// TwinCAT 3 PLC project ThermalControl_PLC
// ProgramVersion: 3.1.4023.0
// libraries:
//   Tc2_ControllerToolbox, * (Beckhoff Automation GmbH)
//   Tc2_Standard, * (Beckhoff Automation GmbH)
//   Tc2_System, * (Beckhoff Automation GmbH)
//   Tc2_TempController, * (Beckhoff Automation GmbH)
//   Tc3_Module, * (Beckhoff Automation GmbH)
// project tree:
//   / Cyclic100ms.TcTTO (not stored), PlcTask.TcTTO
//   DUTs/ E_State.TcDUT (not stored), ST_ThermalCouple.TcDUT (not stored)
//   GVLs/ GVL.TcGVL, HMI_DB.TcGVL (not stored), Input.TcGVL, MCP_IO.TcGVL (not stored), Output.TcGVL
//   POUs/ ADC_10V.TcPOU (not stored), ADC_5V.TcPOU (not stored), Alias.TcPOU, AnalogConversion.TcPOU (not stored), AQ.TcPOU (not stored), AQ_5V.TcPOU, FB_Process.TcPOU, Heartbeat.TcPOU (not stored), MAIN.TcPOU (not stored), Norm_x.TcPOU (not stored), Sequence.TcPOU
//   POUs/Controller/ Controller_v1.TcPOU, Controller_v2.TcPOU (not stored)
//   POUs/PID/ PRG_FB_CTRL_PID.TcPOU

CONFIGURATION ThermalControl_PLC
    RESOURCE PLC ON TwinCAT3
        TASK PlcTask(INTERVAL := T#10ms, PRIORITY := 20);
        PROGRAM MAIN WITH PlcTask : MAIN;
    END_RESOURCE
END_CONFIGURATION

// ---- GVLs/GVL.TcGVL
{attribute 'qualified_only'}
VAR_GLOBAL
	SetpointValueToScope			: LREAL;
	ActualValueToScope				: LREAL;
	OutToScope						: LREAL;
END_VAR

// ---- GVLs/Input.TcGVL
{attribute 'qualified_only'}
VAR_GLOBAL
//***MCP************************************************************************
	//EL3314 - AI1
	R1_01_00 AT	%I*: INT; //Master stop PB not pressed - black pb on mcp
	R1_01_01 AT	%I*: INT; //case Estop circuit okay (Rly1 (120vac)
	R1_01_02 AT %I*: INT; //Remote Mode Selected (NO)
	R1_01_03 AT %I*: INT; //MCP PSU1 DC OK
	
	//EL3314 - AI2
	R1_02_00 AT	%I*: INT; //
	R1_02_01 AT	%I*: INT;
	R1_02_02 AT %I*: INT; 
	R1_02_03 AT %I*: INT; 
	
	//EL3314 - AI3
	R1_03_00 AT	%I*: INT; //
	R1_03_01 AT	%I*: INT;
	R1_03_02 AT %I*: INT; 
	R1_03_03 AT %I*: INT; 

END_VAR

// ---- GVLs/Output.TcGVL
{attribute 'qualified_only'}
VAR_GLOBAL
	//***MCP 
	//EL2008
	R1_13_00 AT %Q*: BOOL;
	
	//EL4008 - AQ1
	R1_18_00 AT %Q*: INT;
	R1_18_01 AT %Q*: INT;
	R1_18_02 AT %Q*: INT;
	R1_18_03 AT %Q*: INT;
	R1_18_04 AT %Q*: INT;
	R1_18_05 AT %Q*: INT;
	R1_18_06 AT %Q*: INT;
	R1_18_07 AT %Q*: INT;

	
END_VAR

// ---- POUs/Alias.TcPOU
PROGRAM Alias
VAR
	i : INT := 0;
END_VAR

 //R1 : MCP**  
	
//INPUT
	//AI	
	MCP_IO.ThermalCouple[1].Temperature_raw					:= Input.R1_01_00;  //NC -
	MCP_IO.ThermalCouple[2].Temperature_raw					:= Input.R1_01_01;  
	MCP_IO.ThermalCouple[3].Temperature_raw					:= Input.R1_01_02; 
	MCP_IO.ThermalCouple[4].Temperature_raw					:= Input.R1_01_03; 

	MCP_IO.ThermalCouple[5].Temperature_raw					:= Input.R1_02_00;  //NC -
	MCP_IO.ThermalCouple[6].Temperature_raw					:= Input.R1_02_01;  
	MCP_IO.ThermalCouple[7].Temperature_raw					:= Input.R1_02_02; 
	MCP_IO.ThermalCouple[8].Temperature_raw					:= Input.R1_02_03; 
	
	MCP_IO.ThermalCouple[9].Temperature_raw					:= Input.R1_03_00;  //NC -
	MCP_IO.ThermalCouple[10].Temperature_raw				:= Input.R1_03_01;  
	MCP_IO.ThermalCouple[11].Temperature_raw				:= Input.R1_03_02; 
	MCP_IO.ThermalCouple[12].Temperature_raw				:= Input.R1_03_03; 
	
	//OUTPUT
	//AQ
	Output.R1_18_00	:= MCP_IO.ChargerSP_raw;
					
	

	
//*************************************************************************************************************

END_PROGRAM

// ---- POUs/AQ_5V.TcPOU
FUNCTION AQ_5V : INT
VAR_INPUT
	Norm_input : REAL;
	x_max : REAL := 10;
	x_min : REAL := 0;
END_VAR
VAR
	voltage_reading : REAL;
END_VAR

voltage_reading := 5 * Norm_input;
AQ_5V := REAL_TO_INT (32767 * (voltage_reading - x_min) / (x_max - x_min));

END_FUNCTION

// ---- POUs/Controller/Controller_v1.TcPOU
PROGRAM Controller_v1

VAR
	
	bOn						: BOOL	:= TRUE;
	bSelSetpoint 			: BOOL	:= FALSE;
	bInit					: BOOL 	:= TRUE;
	bTune					: BOOL 	:= TRUE;
	bManual					: BOOL;

	bNoise 					: BOOL;
	bError 					: BOOL;
	iErrorId 				: E_ErrorCodes;

	fW						: LREAL;						(* setpoint *)
	fW1						: LREAL := 	70;					(* first setpoint *)
	fW2						: LREAL :=	35.0;				(* second setpoint - standby setpoint*)
	fY						: LREAL;						(* control value *)
	fX						: LREAL;						(* actual value from simulated process *)
	bYPWM					: BOOL;

	bSelParameterSet		: BOOL := FALSE;
	bEnableSoftStart 		: BOOL := TRUE;
	bEnableRamping 			: BOOL := FALSE;

	(* parameters *)
	sControllerParameter	:	ST_ControllerParameter := ( 	
	
	iMode 					:= CTRLMODE_HEATING, 							(* 1=heating, 2=cooling, 3=heating&cooling *)
	iReactionOnFailure 		:= TC_OnFailureStopController,					(* 0=controller off, 1=manual op, 2=yMin, 3=yMax *)
	
	dwAlarmSupp 			:= 16#FF_FF_FF_FF, 								(* alarm suppression *)
	tCtrlCycleTime 			:= T#500MS, 									(* controller cycle time *)
	tTaskCycleTime 			:= T#10MS,										(* plc task cycle time *)
	fYTune 					:= 100.0,										(* switch to closed loop control when X > 0.8*W *)
	
	tPWMCycleTime 			:= T#40MS,										(* PWM: period *)
	
	(* setpoint parameters 													 *)	
	fWMin 					:= 0, 											(* lower limit *)
	fWMax 					:= 300,  										(* upper limit *)
	
	(* start up 															*)
	fWStartUp 				:= 0.0, //40.0,									(* soft start plateau setpoint *)
	tStartUp 				:= T#0MS,// T#20S,								(* soft start waiting time*)
 	bStartUpRamping 		:= FALSE,//TRUE, 								(* enable ramping while start up phase *)
	fWStartUpVeloPos 		:= 1.0, 										(* max gradient for increasing setpoint in start up phase*)
	fWStartUpVeloNeg 		:= 1.0,											(* max gradient for decreasing setpoint in start up phase*)
	
	fWVeloPos 				:= 1.0,											(* max gradient for increasing setpoint *) 
	fWVeloNeg 				:= 1.0,											(* max gradient for decreasing setpoint *)	
	
	(* actual value parameters     											 *)	
	bFilter 				:= FALSE, 	
	tFilter 				:= T#0S,
	
	(* control value parameters     										 *)
	fYMin 					:= 0.0, 										(* lower limit *)
	fYMax 					:= 100.0, 										(* upper limit *)
	fYManual 				:= 0.0,											(* manual operation*)
	
	(* controller settings			     									 *)
	bEnablePreController 	:= FALSE,										(* enable precontroller *)		
	bEnableZones 			:= FALSE, 										(* enable zone around setpoint with open loop control *)	
	bEnableCVFilter 		:= FALSE,	 									(* enable filter for CV (type see iFilterType) *)
	iFilterType 			:= E_FilterType_FIRSTORDER,						(* filtertype of CV filter *)
	iControllerType 		:= E_ControllerType_PID,						(* used controller normally PID *)
	
	(* min max temperatures	     											 *)
	TempLow 				:= -5.0, 
	TempLowLow 				:= -10.0,  
	TempHigh			 	:= 5.0, 
	TempHighHigh 			:= 10.0, 
	TempAbsoluteHigh 		:= 300.0, 
	TempAbsoluteLow 		:= 0.0
	
	);
								
	sParaControlExternal	: st_ParaController;
	
	fbTempController		: FB_TempController;
	fbProcess				: FB_Process;
	fbCtrlParameter			: FB_CtrlParameter;	
	
	(* Debug *)
	fMaxOvershoot			: LREAL;
	tStartUpTime			: TIME;
	eCtrlState				: E_CTRL_STATE;	
	
END_VAR

(* Select setpoint *)
IF bSelSetpoint THEN
	fW := fW2;
ELSE
	fW := fW1;
END_IF

(* Simulate process *)
fbProcess(	fY := fbTempController.fYAnalog, 
			bNoise := bNoise, 
			tTa := sControllerParameter.tTaskCycleTime);
			
(* Actual temperature *)				
fX := fbProcess.fX;  // Add measured temperature here

(* Start controller *)
fbTempController(
					bOn						:= bOn,
					bInit					:= bInit,
					bTune					:= bTune,
					bManual					:= bManual,
					bSelSetpoint			:= bSelSetpoint,
					bSelCtrlParameterSet 	:= bSelParameterSet,
					bEnableSoftStart 		:= bEnableSoftStart,
					bEnableRamping 			:= bEnableRamping,
					fW1						:= fW1,
					fW2						:= fW2,
					fX						:= fX,
					bOpenThermocouple		:= FALSE,
					bReverseThermocouple	:= FALSE,
					bBackVoltage			:= FALSE,
					bLeakage				:= FALSE,
					bShortCircuit			:= FALSE,
					bOpenCircuit			:= FALSE,
					sControllerParameter	:= sControllerParameter,
					sParaControllerExternal	:= fbCtrlParameter.sParaController
					);
					
(* Analog output *)			
fY := fbTempController.fYAnalog;
(* Digital (PWM) output *)
bYPWM := fbTempController.bYPWM;

bError := fbTempController.bError;
iErrorId := fbTempController.iErrorId;
bInit := FALSE;	

(* Debug *)
fMaxOvershoot := fbTempController.fMaxOverShoot;
tStartUpTime := fbTempController.tStartUpTime;

(* Scope *)
fW_Scope := fW;
fX_Scope := fX;
fY_Scope := fY;

END_PROGRAM

// ---- POUs/FB_Process.TcPOU
FUNCTION_BLOCK FB_Process

VAR_INPUT
	fY		:	LREAL;
	tTa		:	TIME;
	bNoise	:	BOOL;
END_VAR

VAR_OUTPUT
	fX		:	LREAL;
END_VAR

VAR
	(* Processparameters *)
	tT11		:	TIME	:= t#5s;
	tT12		:	TIME	:= t#25s;

	(* process *)
	fbProcessPart1	:	FB_CTRL_PT1;
	fbProcessPart2	:	FB_CTRL_PT1;
	fbNoise			:	FB_CTRL_NOISE_GENERATOR;

	stProcessPart1	:	ST_CTRL_PT1_PARAMS;
	stProcessPart2	:	ST_CTRL_PT1_PARAMS;
	stNoise			:	ST_CTRL_NOISE_GENERATOR_PARAMS;
	
END_VAR

(* init structures *)
stProcessPart1.fKp := 1.0;
stProcessPart1.tCtrlCycleTime := tTa;
stProcessPart1.tT1 := tT11;
stProcessPart1.tTaskCycleTime := tTa;

stProcessPart2.fKp := 1.0;
stProcessPart2.tCtrlCycleTime := tTa;
stProcessPart2.tT1 := tT12;
stProcessPart2.tTaskCycleTime := tTa;

stNoise.fAmplitude := 1.0;
stNoise.tCtrlCycleTime := tTa;
stNoise.tTaskCycleTime := tTa;

(* calculate and simulate process *)
fbProcessPart1(
				fIn:= fY,
				fManSyncValue:= 0.0,
				bSync:= FALSE,
				eMode:= eCTRL_MODE_ACTIVE,
				bHold:= FALSE,
				stParams:= stProcessPart1);

fbProcessPart2(
				fIn:= fbProcessPart1.fOut,
				fManSyncValue:= 0.0,
				bSync:= FALSE,
				eMode:= eCTRL_MODE_ACTIVE,
				bHold:= FALSE,
				stParams:= stProcessPart2);

fbNoise(
		fManSyncValue:= 0.0,
		eMode:= eCTRL_MODE_ACTIVE,
		stParams:= stNoise);

IF bNoise THEN
	fX := fbProcessPart2.fOut + 0.01*fbNoise.fOut;
ELSE
	fX := fbProcessPart2.fOut;
END_IF;

END_FUNCTION_BLOCK

// ---- POUs/PID/PRG_FB_CTRL_PID.TcPOU
PROGRAM PRG_FB_CTRL_PID
VAR
	SetpointValue				: LREAL		:= 5.0; //setpoint value
	ActualValue					: LREAL;			//feedback signal
	ManSyncValue				: LREAL;			//manual overwrites
	Sync						: BOOL;

	Out							: LREAL;			//output signal
	Hold						: BOOL;
	
// eMode : IDLE = 0, passive = 1, active = 2, reset = 3, manual = 4, tune = 5, selftest = 6, sync movement = 7
// E_CTRL_STATE : IDLE=0, passive=1, active=2, reset=3, manual=4, turning=5, tuned=6, selftest=7, error=8, sync movement =9 
	eMode							: E_CTRL_MODE; //active mode is auto mode, manual mode is manual mode
	eCtrlState						: E_CTRL_STATE;
	CTRL_PID_PARAMS					: ST_CTRL_PID_PARAMS;

	eErrorId						: E_CTRL_ERRORCODES;
	Error							: BOOL;
	ARWactive						: BOOL;

	(* controller *)
	CTRL_PID						: FB_CTRL_PID;

	Init							: BOOL	:= TRUE;
	TON							: TON;
END_VAR

IF Init THEN
	(* init parameter struct *)
	CTRL_PID_PARAMS.tCtrlCycleTime		:= T#500MS;		//contro cycle time
	CTRL_PID_PARAMS.tTaskCycleTime		:= T#100MS;		//task cycle time
	CTRL_PID_PARAMS.fKp					:= 2.0;			(* proportional gain Kp				*)
	CTRL_PID_PARAMS.tTn					:= T#1S;		(*  Tn								*)
	CTRL_PID_PARAMS.tTv					:= T#200MS;		(*  Tv								*)
	CTRL_PID_PARAMS.tTd					:= T#100MS;		(*  Td								*)
	CTRL_PID_PARAMS.fOutMaxLimit			:= 100;			(* maximum output limit				*)
	CTRL_PID_PARAMS.fOutMinLimit			:= 0;			(* minimum output limit				*)

	(* set the mode to ACTIVE --> normal operation *)
	eMode := eCTRL_MODE_ACTIVE;

	(* reset the init flag *)
	Init := FALSE;
END_IF

(*
TYPE E_CTRL_MODE :
(
    eCTRL_MODE_IDLE     := 0, 
    eCTRL_MODE_PASSIVE     := 1, 
    eCTRL_MODE_ACTIVE     := 2, 
    eCTRL_MODE_RESET     := 3, 
    eCTRL_MODE_MANUAL     := 4, 
    eCTRL_MODE_TUNE     := 5, 
    eCTRL_MODE_SELFTEST    := 6, 
    eCTRL_MODE_SYNC_MOVEMENT := 7 
)
END_TYPE

TYPE E_CTRL_STATE :
(
    eCTRL_STATE_IDLE        := 0, 
    eCTRL_STATE_PASSIVE := 1, 
    eCTRL_STATE_ACTIVE := 2, 
    eCTRL_STATE_RESET     := 3, 
    eCTRL_STATE_MANUAL := 4, 
    eCTRL_STATE_TUNING := 5, 
    eCTRL_STATE_TUNED     := 6, 
    eCTRL_STATE_SELFTEST := 7, 
    eCTRL_STATE_ERROR     := 8, 
    eCTRL_STATE_SYNC_MOVEMENT := 9 
);
END_TYPE
*)

SetpointValue := HMI_DB.TemperatureSP; //setpoint
ActualValue := Sequence.AverageTemp; //feedback

MCP_IO.ChargerSP := Out; //output

(* copy var to scope var *)
GVL.SetpointValueToScope 	:= SetpointValue;
GVL.ActualValueToScope 		:= ActualValue;


(* call controller *)
CTRL_PID(		fSetpointValue		:= SetpointValue, //setpoint value
				fActualValue		:= ActualValue, //temperature average fd value (analog input scaled value)
				fManSyncValue		:= ManSyncValue, // if stop heater, manual mode takes over and set the sp to 0- basically manual output (0-100)
				bSync				:= Sync,
				eMode				:= eMode,
				bHold				:= Hold,
				stParams			:= CTRL_PID_PARAMS,
				fOut				=> Out, //control signal - analog output value
				bARWactive			=> ARWactive,
				eErrorId			=> eErrorId,
				bError				=> Error
				);


(* copy var to scope var *)
GVL.OutToScope := Out;

END_PROGRAM

// ---- POUs/Sequence.TcPOU
PROGRAM Sequence  //make sure the change the name to Sequence when we use it for the HMI bitmappings.
VAR
	AverageTemp		: REAL := 0;
	Sum				: REAL := 0;;
	i				: INT := 1;
	n				: INT := 12;
	NumOfTherm		: UINT := 12;
END_VAR


//find sum
FOR i := 1 TO n BY 1 DO 
	
	Sum := Sum + MCP_IO.ThermalCouple[i].TemperatureFB;

END_FOR
	
NumOfTherm.0 := HMI_DB.ThermalCouple[1].IncludeSW;
NumOfTherm.1 := HMI_DB.ThermalCouple[2].IncludeSW;
NumOfTherm.2 := HMI_DB.ThermalCouple[3].IncludeSW;
NumOfTherm.3 := HMI_DB.ThermalCouple[4].IncludeSW;
NumOfTherm.4 := HMI_DB.ThermalCouple[5].IncludeSW;
NumOfTherm.5 := HMI_DB.ThermalCouple[6].IncludeSW;
NumOfTherm.6 := HMI_DB.ThermalCouple[7].IncludeSW;
NumOfTherm.7 := HMI_DB.ThermalCouple[8].IncludeSW;
NumOfTherm.8 := HMI_DB.ThermalCouple[9].IncludeSW;
NumOfTherm.9 := HMI_DB.ThermalCouple[10].IncludeSW;
NumOfTherm.10 := HMI_DB.ThermalCouple[11].IncludeSW;
NumOfTherm.11 := HMI_DB.ThermalCouple[12].IncludeSW;


//USED AS FEEDBACK
AverageTemp := Sum/NumOfTherm;



//PRG_FB_CTRL_PID();


IF i > n THEN
	i := 1;
END_IF

END_PROGRAM
